Staubli VAL3: io.pjx

--- io.pjx ---
Parameters version=s7.8.3 stackSize=5000 millimeterUnit=true
Program file=start.pgx
Program file=stop.pgx
Data file=io.dtx

--- io.dtx ---
mdesc mNomSpeed
public dio dInCrashError = {link=ApplicomIO-1\TOPIC1_A-BLOCKA\%I0[0]}
public dio dOutIsReady = {link=ApplicomIO-1\TOPIC1_A-BLOCKA\%Q0[5]}
public string sToShow
public dio dInStart = {link=ApplicomIO-1\TOPIC1_A-BLOCKA\%I0[0]}
public dio dInStop
